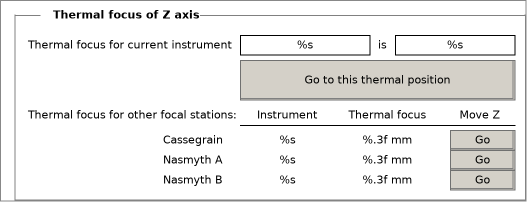
VISUALIZATION VISU_M2ThermalFocus  // 527x202
VAR_IN_OUT
	ref : M2;
    widget : M2Widget;
END_VAR
    Polyline (200,15) (525,15) (525,200) (15,200) (15,15) (40,15)
    Label (25,35 210x20), "Thermal focus for current instrument"
    Label (50,5 150x20), "Thermal focus of Z axis"
    Rectangle (240,35 130x20), "%s", text variable: widget.actualFocalStationName
    Label (375,35 25x20), "is"
    Rectangle (395,35 120x20), "%s", text variable: widget.actualFocalStationThermalFocus
    Button (240,60 275x40), "Go to this thermal position", input disabled if: ref.processes.doThermalFocus.statuses.enabledStatus.disabled
        OnMouseClick: execute { ref.processes.doThermalFocus.do_request := TRUE; }
    Label (25,105 220x20), "Thermal focus for other focal stations:"
    Button (450,130 65x20), "Go", input disabled if: ref.processes.doThermalFocusForStationPosition.statuses.enabledStatus.disabled
        OnMouseClick: execute { ref.processes.doThermalFocusForStationPosition.set.station := M3PositionIDs.CASSEGRAIN; ref.processes.doThermalFocusForStationPosition.do_request := TRUE; }
    Rectangle (240,130 95x20), "%s", text variable: widget.cassegrainName
    Label (160,130 80x20), "Cassegrain"
    Rectangle (345,130 85x20), "%.3f mm", text variable: ref.thermalFocusCassegrain.millimeters.value
    Line (240,125) (515,125)
    Label (240,105 95x20), "Instrument"
    Label (345,105 85x20), "Thermal focus"
    Label (445,105 70x20), "Move Z"
    Rectangle (240,150 95x20), "%s", text variable: widget.nasmythAName
    Label (160,150 80x20), "Nasmyth A"
    Rectangle (345,150 85x20), "%.3f mm", text variable: ref.thermalFocusNasmythA.millimeters.value
    Rectangle (240,170 95x20), "%s", text variable: widget.nasmythBName
    Label (160,170 80x20), "Nasmyth B"
    Rectangle (345,170 85x20), "%.3f mm", text variable: ref.thermalFocusNasmythB.millimeters.value
    Button (450,150 65x20), "Go", input disabled if: ref.processes.doThermalFocusForStationPosition.statuses.enabledStatus.disabled
        OnMouseClick: execute { ref.processes.doThermalFocusForStationPosition.set.station := M3PositionIDs.NASMYTH_A; ref.processes.doThermalFocusForStationPosition.do_request := TRUE; }
    Button (450,170 65x20), "Go", input disabled if: ref.processes.doThermalFocusForStationPosition.statuses.enabledStatus.disabled
        OnMouseClick: execute { ref.processes.doThermalFocusForStationPosition.set.station := M3PositionIDs.NASMYTH_B; ref.processes.doThermalFocusForStationPosition.do_request := TRUE; }
END_VISUALIZATION

(* stored: Version 1.1.0.1, ProductVersion 3.1.4019.2
   Visu VISU_M2ThermalFocus: Id {5b5ddf7c-3b4a-463c-85dc-ffb47f275907} *)
